FUNCTION_BLOCK FB_MyUpCounter
VAR_INPUT
    // Count up signal
    CU: BOOL;
END_VAR
VAR_OUTPUT
    // Current cunter value output
    CV: INT;
END_VAR
VAR
    // Count is up in current cycle
    bLastCount: BOOL;
END_VAR

IF NOT bLastCount AND CU THEN
    CV := CV + 1;
END_IF

// Set flag to TRUE if count is increased in current cycle
bLastCount := CU;

END_FUNCTION_BLOCK

(* stored: Version 1.1.0.1
   POU FB_MyUpCounter: Id {b814e1b6-7e75-48af-87c0-eef03af6b5bf}, SpecialFunc None *)
